{attribute addProperty BoxType "EP5101-2011-0016"}
{attribute addProperty Id "ENC_Status_compactAT %I*ENC_Status_compact_6BB1ED4B4860ENC_Control_compactAT %Q*ENC_Control_compact_03701F333240WcStateAT %I*WcState_F855686C1620InfoDataAT %I*InfoData_BC63D37F80100"}
{attribute addProperty CRC "4234364568"}
{attribute addProperty SizeInBites "176"}
{attribute addProperty SizeInBytes "22"}
TYPE EP5101_22B069AD :
STRUCT
	{attribute addProperty Name "ENC_Status_compact"}
	ENC_Status_compact : ENC_Status_compact_6BB1ED4B;
	{attribute addProperty Name "ENC_Control_compact"}
	ENC_Control_compact : ENC_Control_compact_03701F33;
	{attribute addProperty Name "WcState"}
	WcState : WcState_F855686C;
	{attribute addProperty Name "InfoData"}
	InfoData : InfoData_BC63D37F;
END_STRUCT
END_TYPE

(* stored: Version 1.2.0.0, ProductVersion 3.1.4024.9
   DUT EP5101_22B069AD: Id {3976644c-ff0b-4aff-b170-f6f16dfdd317} *)
